(* PLC project SafeLOGIC-1, BrAutomation SafeDESIGNER  4.3.4.4 *)
(* stored: companyURL http://www.br-automation.com, creationDateTime Thu Jun 24 15:32:52 2021 *)

PROGRAM Main
  VAR  (* added by the conversion: wires and edge detectors of the diagram *)
    _SAFEBOOL_TO_BOOL118_OUT : BOOL;
  END_VAR

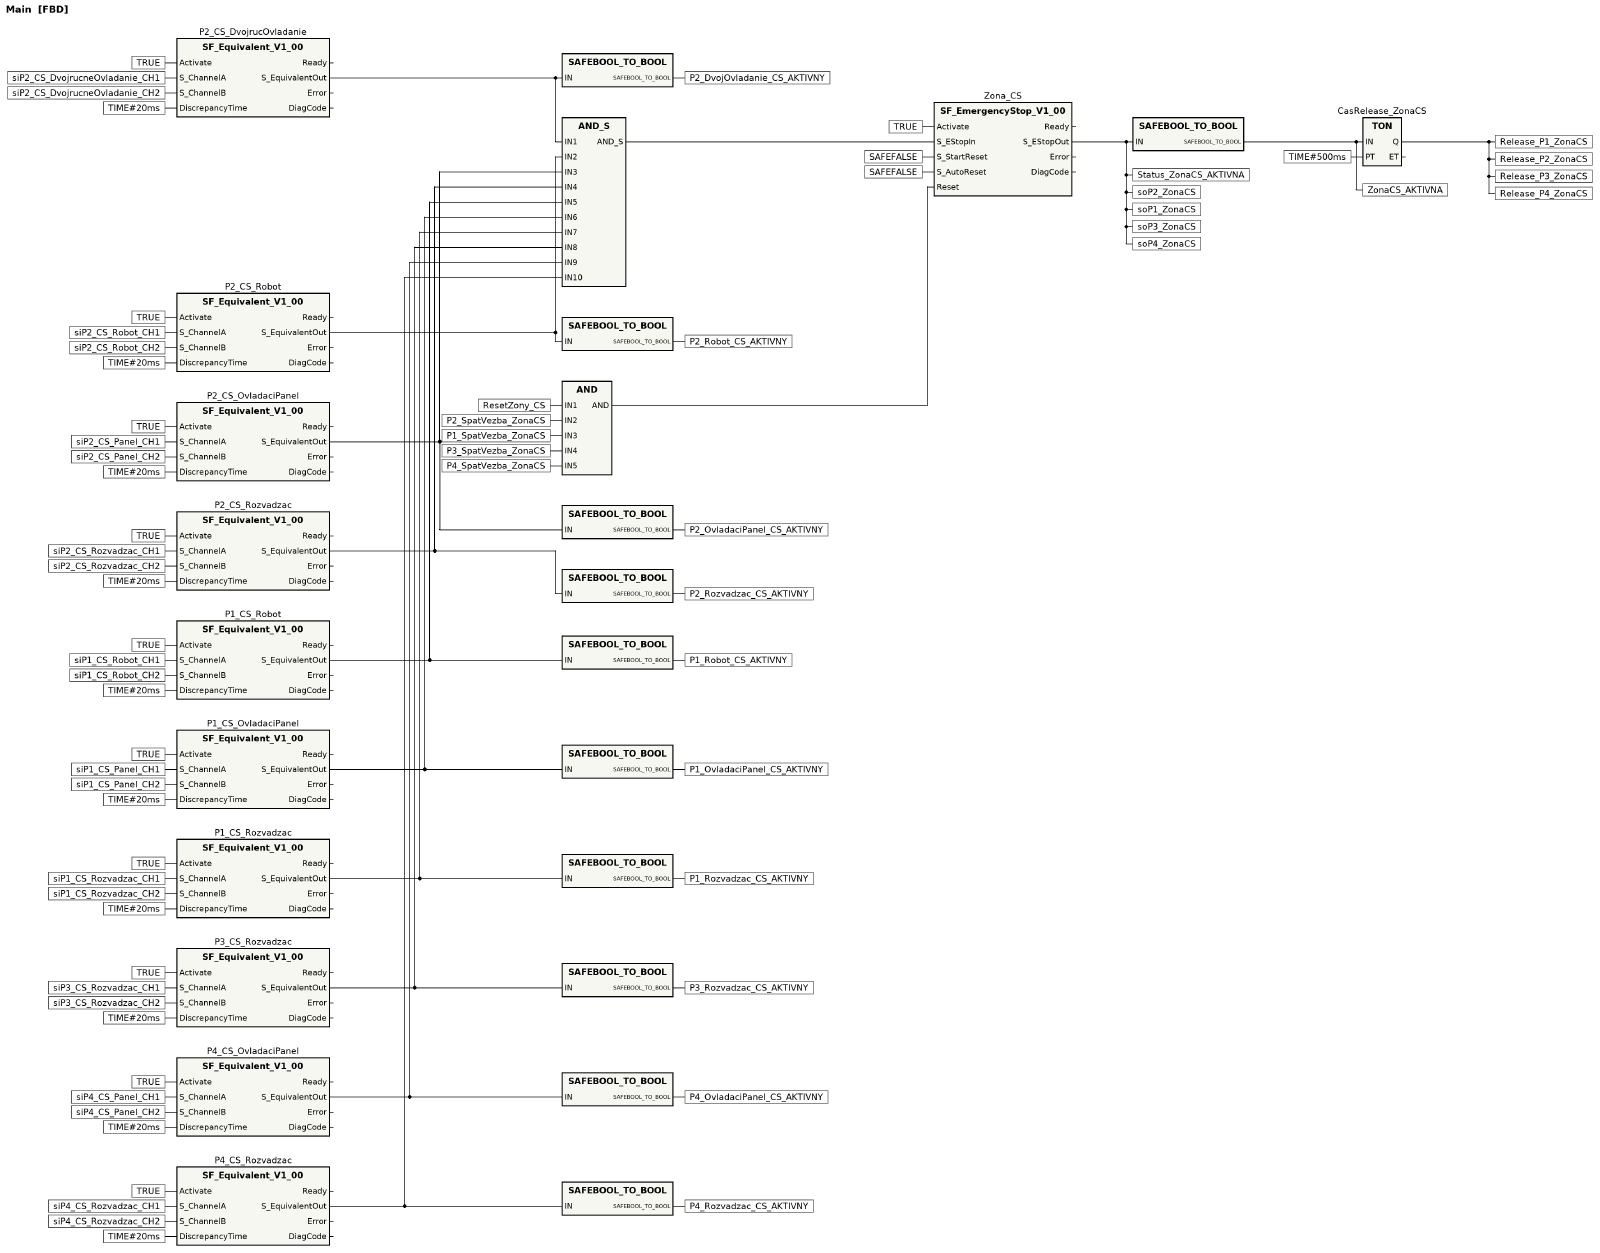
(* FBD diagram, written out as Structured Text *)
P2_CS_DvojrucOvladanie(Activate := TRUE, S_ChannelA := siP2_CS_DvojrucneOvladanie_CH1, S_ChannelB := siP2_CS_DvojrucneOvladanie_CH2, DiscrepancyTime := TIME#20ms);
P2_CS_Robot(Activate := TRUE, S_ChannelA := siP2_CS_Robot_CH1, S_ChannelB := siP2_CS_Robot_CH2, DiscrepancyTime := TIME#20ms);
P2_CS_OvladaciPanel(Activate := TRUE, S_ChannelA := siP2_CS_Panel_CH1, S_ChannelB := siP2_CS_Panel_CH2, DiscrepancyTime := TIME#20ms);
P2_CS_Rozvadzac(Activate := TRUE, S_ChannelA := siP2_CS_Rozvadzac_CH1, S_ChannelB := siP2_CS_Rozvadzac_CH2, DiscrepancyTime := TIME#20ms);
P1_CS_Robot(Activate := TRUE, S_ChannelA := siP1_CS_Robot_CH1, S_ChannelB := siP1_CS_Robot_CH2, DiscrepancyTime := TIME#20ms);
P1_CS_OvladaciPanel(Activate := TRUE, S_ChannelA := siP1_CS_Panel_CH1, S_ChannelB := siP1_CS_Panel_CH2, DiscrepancyTime := TIME#20ms);
P1_CS_Rozvadzac(Activate := TRUE, S_ChannelA := siP1_CS_Rozvadzac_CH1, S_ChannelB := siP1_CS_Rozvadzac_CH2, DiscrepancyTime := TIME#20ms);
P3_CS_Rozvadzac(Activate := TRUE, S_ChannelA := siP3_CS_Rozvadzac_CH1, S_ChannelB := siP3_CS_Rozvadzac_CH2, DiscrepancyTime := TIME#20ms);
P4_CS_OvladaciPanel(Activate := TRUE, S_ChannelA := siP4_CS_Panel_CH1, S_ChannelB := siP4_CS_Panel_CH2, DiscrepancyTime := TIME#20ms);
P4_CS_Rozvadzac(Activate := TRUE, S_ChannelA := siP4_CS_Rozvadzac_CH1, S_ChannelB := siP4_CS_Rozvadzac_CH2, DiscrepancyTime := TIME#20ms);
Zona_CS(Activate := TRUE, S_EStopIn := AND_S(P2_CS_DvojrucOvladanie.S_EquivalentOut, P2_CS_Robot.S_EquivalentOut, P2_CS_OvladaciPanel.S_EquivalentOut, P2_CS_Rozvadzac.S_EquivalentOut, P1_CS_Robot.S_EquivalentOut, P1_CS_OvladaciPanel.S_EquivalentOut, P1_CS_Rozvadzac.S_EquivalentOut, P3_CS_Rozvadzac.S_EquivalentOut, P4_CS_OvladaciPanel.S_EquivalentOut, P4_CS_Rozvadzac.S_EquivalentOut), S_StartReset := SAFEFALSE, S_AutoReset := SAFEFALSE, Reset := ResetZony_CS AND P2_SpatVezba_ZonaCS AND P1_SpatVezba_ZonaCS AND P3_SpatVezba_ZonaCS AND P4_SpatVezba_ZonaCS);
soP2_ZonaCS := Zona_CS.S_EStopOut;
P2_DvojOvladanie_CS_AKTIVNY := SAFEBOOL_TO_BOOL(P2_CS_DvojrucOvladanie.S_EquivalentOut);
soP1_ZonaCS := Zona_CS.S_EStopOut;
soP3_ZonaCS := Zona_CS.S_EStopOut;
soP4_ZonaCS := Zona_CS.S_EStopOut;
Status_ZonaCS_AKTIVNA := Zona_CS.S_EStopOut;
P2_Robot_CS_AKTIVNY := SAFEBOOL_TO_BOOL(P2_CS_Robot.S_EquivalentOut);
_SAFEBOOL_TO_BOOL118_OUT := SAFEBOOL_TO_BOOL(Zona_CS.S_EStopOut);
ZonaCS_AKTIVNA := _SAFEBOOL_TO_BOOL118_OUT;
CasRelease_ZonaCS(IN := _SAFEBOOL_TO_BOOL118_OUT, PT := TIME#500ms);
Release_P1_ZonaCS := CasRelease_ZonaCS.Q;
Release_P2_ZonaCS := CasRelease_ZonaCS.Q;
Release_P3_ZonaCS := CasRelease_ZonaCS.Q;
Release_P4_ZonaCS := CasRelease_ZonaCS.Q;
P2_OvladaciPanel_CS_AKTIVNY := SAFEBOOL_TO_BOOL(P2_CS_OvladaciPanel.S_EquivalentOut);
P2_Rozvadzac_CS_AKTIVNY := SAFEBOOL_TO_BOOL(P2_CS_Rozvadzac.S_EquivalentOut);
P1_Robot_CS_AKTIVNY := SAFEBOOL_TO_BOOL(P1_CS_Robot.S_EquivalentOut);
P1_OvladaciPanel_CS_AKTIVNY := SAFEBOOL_TO_BOOL(P1_CS_OvladaciPanel.S_EquivalentOut);
P1_Rozvadzac_CS_AKTIVNY := SAFEBOOL_TO_BOOL(P1_CS_Rozvadzac.S_EquivalentOut);
P3_Rozvadzac_CS_AKTIVNY := SAFEBOOL_TO_BOOL(P3_CS_Rozvadzac.S_EquivalentOut);
P4_OvladaciPanel_CS_AKTIVNY := SAFEBOOL_TO_BOOL(P4_CS_OvladaciPanel.S_EquivalentOut);
P4_Rozvadzac_CS_AKTIVNY := SAFEBOOL_TO_BOOL(P4_CS_Rozvadzac.S_EquivalentOut);
END_PROGRAM
